Fanuc TP program (LS listing): MTCOUNT.printtp.LS

/PROG  MTCOUNT
/ATTR
OWNER		= MNEDITOR;
COMMENT		= "MtCount         ";
PROG_SIZE	= 234;
CREATE		= DATE 26-10-06  TIME 16:17:00;
MODIFIED	= DATE 26-10-06  TIME 16:17:00;
FILE_NAME	= ;
VERSION		= 0;
LINE_COUNT	= 2;
MEMORY_SIZE	= 598;
PROTECT		= READ_WRITE;
TCD:  STACK_SIZE	= 0,
      TASK_PRIORITY	= 50,
      TIME_SLICE	= 0,
      BUSY_LAMP_OFF	= 0,
      ABORT_REQUEST	= 0,
      PAUSE_REQUEST	= 0;
DEFAULT_GROUP	= 1,*,*,*,*;
CONTROL_CODE	= 00000000 00000000;
LOCAL_REGISTERS	= 0,0,0;
/MN
   1:  !RAPID MakeTpProbe.MtCount ;
   2:  R[2:mtCalls]=R[2:mtCalls]+1    ;
/POS
/END
